Universal Robots PolyScope program: iniciales1-nombres_NEW.urp

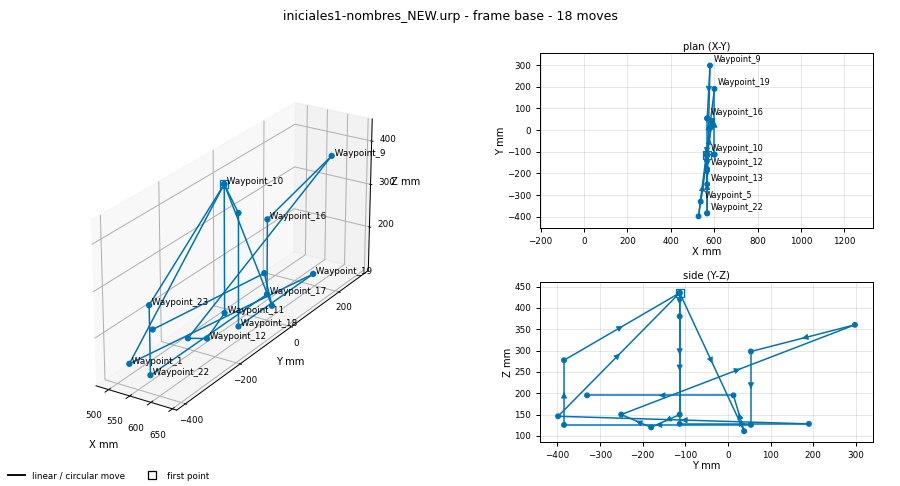
[picture p0: tool path of iniciales1-nombres_NEW.urp in frame base, 18 of 18 moves have a stored position in this frame; points joined in program order, loops and branches not executed]
Program iniciales1-nombres (installation=default directory=/ursim/programs createdIn=3.15.8.106339 lastSavedIn=3.15.8.106339 robotSerialNumber=2018359999)
Calibrated DH parameters: a=[0, -0.425, -0.39225, 0, 0, 0]; d=[0.089159, 0, 0, 0.10915, 0.09465, 0.0823]; alpha=[1.570796, 0, 0, 1.570796, -1.570796, 0]; deltaTheta=[0, 0, 0, 0, 0, 0]
Robot Program (runOnlyOnce=false)
  Popup Message (haltProgram=false message=se va a realizar la letra J inputType=Text)
  MoveL speed 250 mm/s, acceleration 1200 mm/s^2 (useActiveTCP=true) feature=Base
    Waypoint Waypoint_10: TCP in base x=568 y=-113 z=435 mm, rx=-0.0012 ry=3.1163 rz=0.0389 rad; joints [-0.597, -161.353, 30.024, 42.751, -91.445, -90.624] deg
    Wait Sleep waitTime=0.5
    Waypoint Waypoint_11: TCP in base x=568 y=-113 z=150 mm, rx=-0.0012 ry=3.1163 rz=0.0389 rad; joints [-0.597, -200.087, 68.065, 43.443, -91.445, -90.624] deg
    Wait Sleep waitTime=0.5
    Waypoint Waypoint_12: TCP in base x=568 y=-180 z=120 mm, rx=-0.0012 ry=3.1163 rz=0.0389 rad; joints [-7.253, -201.508, 65.201, 47.551, -91.6, -97.28] deg
    Wait Sleep waitTime=0.5
    Waypoint Waypoint_13: TCP in base x=568 y=-250 z=150 mm, rx=-0.0012 ry=3.1163 rz=0.0389 rad; joints [-13.86, -195.521, 56.757, 49.816, -91.733, -103.889] deg
  Popup Message (haltProgram=false message=se va a realizar la letra G inputType=Text)
  MoveL speed 250 mm/s, acceleration 1200 mm/s^2 (useActiveTCP=true) feature=Base
    Waypoint Waypoint_9: TCP in base x=580.883 y=297.633 z=360.302 mm, rx=-0.0247 ry=3.1164 rz=0.0392 rad; joints [36.716, -154.128, 0.014, 66.116, -90.318, -54.186] deg
    Wait Sleep waitTime=0.5
    Waypoint Waypoint_16: TCP in base x=568 y=53.921 z=297.802 mm, rx=-0.0012 ry=3.1163 rz=0.0389 rad; joints [16.31, -183.411, 57.856, 37.335, -90.969, -73.72] deg
    Wait Sleep waitTime=0.5
    Waypoint Waypoint_17: TCP in base x=568 y=53.921 z=125.803 mm, rx=-0.0012 ry=3.1163 rz=0.0389 rad; joints [16.31, -203.51, 71.481, 43.809, -90.969, -73.72] deg
    Wait Sleep waitTime=0.5
    Waypoint Waypoint_22: TCP in base x=568 y=-384.075 z=125.803 mm, rx=-0.0012 ry=3.1163 rz=0.0389 rad; joints [-25.138, -187.746, 34.621, 63.817, -91.905, -115.171] deg
    Wait Sleep waitTime=0.5
    Waypoint Waypoint_23: TCP in base x=567.825 y=-383.993 z=277.31 mm, rx=-0.0012 ry=3.1163 rz=0.0389 rad; joints [-25.138, -160.403, -0.398, 71.493, -91.905, -115.171] deg
    Wait Sleep waitTime=0.5
    Waypoint Waypoint_24: TCP in base x=568 y=-113 z=435 mm, rx=-0.0012 ry=3.1163 rz=0.0389 rad; joints [-0.597, -161.353, 30.024, 42.751, -91.445, -90.624] deg
  Popup Message (haltProgram=false message=se va a realizar la letra L inputType=Text)
  MoveL speed 250 mm/s, acceleration 1200 mm/s^2 (useActiveTCP=true) feature=Base
    Waypoint Waypoint_8: TCP in base x=601.465 y=-112.989 z=380.153 mm, rx=-0.0012 ry=3.1163 rz=0.0389 rad; joints [-0.563, -165.83, 29.641, 47.611, -91.444, -90.59] deg
    Wait Sleep waitTime=0.5
    Waypoint Waypoint_18: TCP in base x=601.465 y=-112.989 z=128.156 mm, rx=-0.0012 ry=3.1163 rz=0.0389 rad; joints [-0.563, -198.847, 60.538, 49.732, -91.444, -90.59] deg
    Wait Sleep waitTime=0.5
    Waypoint Waypoint_19: TCP in base x=601.465 y=189.809 z=128.156 mm, rx=-0.0012 ry=3.1163 rz=0.0389 rad; joints [27.4, -196.57, 55.343, 53.16, -90.609, -62.635] deg
  Popup Message (haltProgram=false message=se va a realizar la letra A inputType=Text)
  MoveL speed 250 mm/s, acceleration 1200 mm/s^2 (useActiveTCP=true) feature=Base
    Waypoint Waypoint_1: TCP in base x=528 y=-398 z=146 mm, rx=-0.0392 ry=2.2037 rz=-2.2037 rad; joints [138.719, -36.697, 84.759, -228.062, -136.695, -0.012] deg
    Wait Sleep waitTime=0.5
    Waypoint Waypoint_2: TCP in base x=568 y=-113 z=435 mm, rx=-0.0392 ry=2.2037 rz=-2.2037 rad; joints [165.765, -64.103, 83.633, -199.53, -163.741, -0.013] deg
    Wait Sleep waitTime=0.5
    Waypoint Waypoint_3: TCP in base x=590 y=38 z=111 mm, rx=-0.0392 ry=2.2037 rz=-2.2037 rad; joints [181.081, -34.231, 86.897, -232.669, -179.057, -0.015] deg
    Wait Sleep waitTime=0.5
    Waypoint Waypoint_4: TCP in base x=586 y=13 z=195 mm, rx=-0.0392 ry=2.2037 rz=-2.2037 rad; joints [178.631, -43.588, 89.519, -225.932, -176.607, -0.013] deg
    Wait Sleep waitTime=0.5
    Waypoint Waypoint_5: TCP in base x=538 y=-330 z=195 mm, rx=-0.0392 ry=2.2037 rz=-2.2037 rad; joints [144.488, -43.698, 89.754, -226.056, -142.465, -0.012] deg
